// Mitsubishi GX Works2 project: Test Output Coil   PLC: FX1N/FX1NC

PROGRAM MAIN
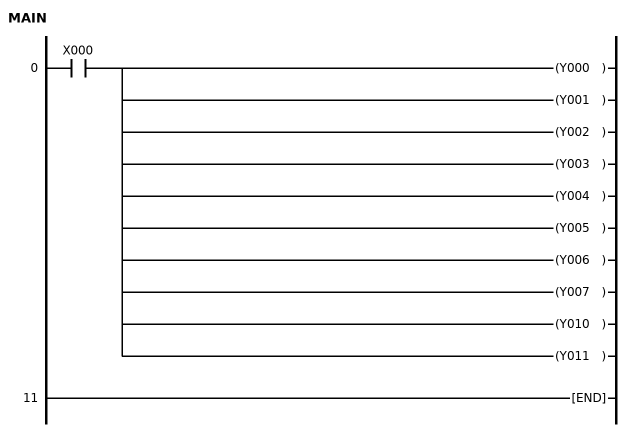
0     LD      X000
      OUT     Y000
      OUT     Y001
      OUT     Y002
      OUT     Y003
      OUT     Y004
      OUT     Y005
      OUT     Y006
      OUT     Y007
      OUT     Y010
      OUT     Y011
11    END
END_PROGRAM
